LIN {X 0,Y 189.818,Z 500.496,A -85,B 0,C 180,E1 4850.971,E2 4850.971} C_VEL
LIN {X 0,Y 177.426,Z 516.785,A -85,B 0,C 180,E1 4849.524,E2 4849.524} C_VEL
LIN {X 0,Y 163.744,Z 531.874,A -85,B 0,C 180,E1 4847.674,E2 4847.674} C_VEL
LIN {X 0,Y 148.865,Z 545.693,A -85,B 0,C 180,E1 4845.27,E2 4845.27} C_VEL
LIN {X 0,Y 133.387,Z 557.829,A -85,B 0,C 180,E1 4842.163,E2 4842.163} C_VEL
LIN {X 0,Y 117.507,Z 568.332,A -85,B 0,C 180,E1 4838.035,E2 4838.035} C_VEL
LIN {X 0,Y 101.557,Z 577.191,A -85,B 0,C 180,E1 4832.376,E2 4832.376} C_VEL
LIN {X 0,Y 86.866,Z 584.067,A -85,B 0,C 180,E1 4824.801,E2 4824.801} C_VEL
LIN {X 0,Y 73.302,Z 589.412,A -85,B 0,C 180,E1 4813.7,E2 4813.7} C_VEL
LIN {X 0,Y 63.497,Z 592.778,A -85,B 0,C 180,E1 4799.212,E2 4799.212} C_VEL
LIN {X 0,Y 58.16,Z 594.477,A -85,B 0,C 180,E1 4780.894,E2 4780.894} C_VEL
LIN {X 0,Y 57.57,Z 594.636,A -85,B 0,C 180,E1 4765.012,E2 4765.012} C_VEL
LIN {X 0,Y 61.019,Z 593.564,A -85,B 0,C 180,E1 4746.836,E2 4746.836} C_VEL
LIN {X 0,Y 68.986,Z 590.981,A -85,B 0,C 180,E1 4731.442,E2 4731.442} C_VEL
LIN {X 0,Y 79.249,Z 587.223,A -85,B 0,C 180,E1 4720.526,E2 4720.526} C_VEL
LIN {X 0,Y 61.349,Z 590.587,A -85,B 0,C 180,E1 4687.494,E2 4687.494} C_VEL
LIN {X 0,Y 60.347,Z 592.025,A -85,B 0,C 180,E1 4673.342,E2 4673.342} C_VEL
LIN {X 0,Y 62.82,Z 593.696,A -85,B 0,C 180,E1 4658.528,E2 4658.528} C_VEL
LIN {X 0,Y 72.454,Z 596.219,A -85,B 0,C 180,E1 4640.504,E2 4640.504} C_VEL
LIN {X 0,Y 61.913,Z 600.596,A -85,B 0,C 180,E1 4625.554,E2 4625.554} C_VEL
LIN {X 0,Y 56.913,Z 603.196,A -85,B 0,C 180,E1 4606.332,E2 4606.332} C_VEL
LIN {X 0,Y 57.134,Z 603.987,A -85,B 0,C 180,E1 4591.009,E2 4591.009} C_VEL
LIN {X 0,Y 56.697,Z 603.74,A -85,B 0,C 180,E1 4581.896,E2 4581.896} C_VEL
LIN {X 0,Y 58.725,Z 601.943,A -85,B 0,C 180,E1 4562.639,E2 4562.639} C_VEL
LIN {X 0,Y 66.617,Z 598.284,A -85,B 0,C 180,E1 4545.144,E2 4545.144} C_VEL
LIN {X 0,Y 79.052,Z 592.754,A -85,B 0,C 180,E1 4532.077,E2 4532.077} C_VEL
LIN {X 0,Y 93.56,Z 585.667,A -85,B 0,C 180,E1 4523.221,E2 4523.221} C_VEL
LIN {X 0,Y 108.939,Z 577.083,A -85,B 0,C 180,E1 4517.079,E2 4517.079} C_VEL
LIN {X 0,Y 124.062,Z 567.359,A -85,B 0,C 180,E1 4512.807,E2 4512.807} C_VEL
LIN {X 0,Y 139.915,Z 555.487,A -85,B 0,C 180,E1 4509.459,E2 4509.459} C_VEL
LIN {X 0,Y 155.122,Z 542.173,A -85,B 0,C 180,E1 4506.984,E2 4506.984} C_VEL
LIN {X 0,Y 169.889,Z 526.958,A -85,B 0,C 180,E1 4505.064,E2 4505.064} C_VEL
LIN {X 0,Y 177.913,Z 517.465,A -85,B 0,C 180,E1 4504.176,E2 4504.176} C_VEL
LIN {X 0,Y 182.355,Z 511.668,A -85,B 0,C 180,E1 4503.395,E2 4503.395} C_VEL
LIN {X 0,Y 192.382,Z 496.615,A -85,B 0,C 180,E1 4500.658,E2 4500.658} C_VEL
LIN {X 0,Y 196.325,Z 490.237,A -85,B 0,C 180,E1 4500.079,E2 4500.079} C_VEL
LIN {X 0,Y 206.249,Z 472.484,A -85,B 0,C 180,E1 4499.444,E2 4499.444} C_VEL
LIN {X 0,Y 214.496,Z 454.315,A -85,B 0,C 180,E1 4498.981,E2 4498.981} C_VEL
LIN {X 0,Y 221.368,Z 434.904,A -85,B 0,C 180,E1 4498.629,E2 4498.629} C_VEL
LIN {X 0,Y 226.556,Z 414.734,A -85,B 0,C 180,E1 4498.331,E2 4498.331} C_VEL
LIN {X 0,Y 230.027,Z 393.555,A -85,B 0,C 180,E1 4498.043,E2 4498.043} C_VEL
LIN {X 0,Y 234.56,Z 356.946,A -85,B 0,C 180,E1 4497.556,E2 4497.556} C_VEL
LIN {X 0,Y 234.539,Z 357.104,A -85,B 0,C 180,E1 4497.279,E2 4497.279} C_VEL
LIN {X 0,Y 228.09,Z 406.713,A -85,B 0,C 180,E1 4496.629,E2 4496.629} C_VEL
LIN {X 0,Y 223.651,Z 426.828,A -85,B 0,C 180,E1 4496.277,E2 4496.277} C_VEL
LIN {X 0,Y 217.544,Z 446.236,A -85,B 0,C 180,E1 4495.807,E2 4495.807} C_VEL
LIN {X 0,Y 209.702,Z 465.163,A -85,B 0,C 180,E1 4495.188,E2 4495.188} C_VEL
LIN {X 0,Y 199.927,Z 483.847,A -85,B 0,C 180,E1 4494.376,E2 4494.376} C_VEL
LIN {X 0,Y 188.732,Z 501.277,A -85,B 0,C 180,E1 4493.36,E2 4493.36} C_VEL
LIN {X 0,Y 176.15,Z 517.521,A -85,B 0,C 180,E1 4492.076,E2 4492.076} C_VEL
LIN {X 0,Y 162.227,Z 532.577,A -85,B 0,C 180,E1 4490.432,E2 4490.432} C_VEL
LIN {X 0,Y 147.978,Z 545.6,A -85,B 0,C 180,E1 4488.432,E2 4488.432} C_VEL
LIN {X 0,Y 132.08,Z 557.864,A -85,B 0,C 180,E1 4485.678,E2 4485.678} C_VEL
LIN {X 0,Y 115.647,Z 568.483,A -85,B 0,C 180,E1 4481.985,E2 4481.985} C_VEL
LIN {X 0,Y 98.949,Z 577.451,A -85,B 0,C 180,E1 4476.849,E2 4476.849} C_VEL
LIN {X 0,Y 82.499,Z 584.718,A -85,B 0,C 180,E1 4469.363,E2 4469.363} C_VEL
LIN {X 0,Y 67.953,Z 589.994,A -85,B 0,C 180,E1 4458.617,E2 4458.617} C_VEL
LIN {X 0,Y 56.638,Z 593.427,A -85,B 0,C 180,E1 4443.171,E2 4443.171} C_VEL
LIN {X 0,Y 50.342,Z 595.123,A -85,B 0,C 180,E1 4422.612,E2 4422.612} C_VEL
LIN {X 0,Y 49.628,Z 595.281,A -85,B 0,C 180,E1 4404.211,E2 4404.211} C_VEL
LIN {X 0,Y 53.752,Z 594.211,A -85,B 0,C 180,E1 4383.478,E2 4383.478} C_VEL
LIN {X 0,Y 63.506,Z 591.436,A -85,B 0,C 180,E1 4366.144,E2 4366.144} C_VEL
LIN {X 0,Y 68.796,Z 589.752,A -85,B 0,C 180,E1 4360.217,E2 4360.217} C_VEL
LIN {X 0,Y 53.866,Z 592.475,A -85,B 0,C 180,E1 4329.619,E2 4329.619} C_VEL
LIN {X 0,Y 52.595,Z 594.013,A -85,B 0,C 180,E1 4312.355,E2 4312.355} C_VEL
LIN {X 0,Y 55.296,Z 595.519,A -85,B 0,C 180,E1 4296.561,E2 4296.561} C_VEL
LIN {X 0,Y 62.782,Z 597.31,A -85,B 0,C 180,E1 4281.136,E2 4281.136} C_VEL
LIN {X 0,Y 52.465,Z 601.062,A -85,B 0,C 180,E1 4263.559,E2 4263.559} C_VEL
LIN {X 0,Y 48.69,Z 603.014,A -85,B 0,C 180,E1 4241.858,E2 4241.858} C_VEL
LIN {X 0,Y 49.2,Z 603.359,A -85,B 0,C 180,E1 4230.007,E2 4230.007} C_VEL
LIN {X 0,Y 48.989,Z 602.601,A -85,B 0,C 180,E1 4212.181,E2 4212.181} C_VEL
LIN {X 0,Y 54.226,Z 600.219,A -85,B 0,C 180,E1 4191.186,E2 4191.186} C_VEL
LIN {X 0,Y 64.861,Z 596.198,A -85,B 0,C 180,E1 4175.224,E2 4175.224} C_VEL
LIN {X 0,Y 79.729,Z 590.089,A -85,B 0,C 180,E1 4163.739,E2 4163.739} C_VEL
LIN {X 0,Y 95.858,Z 582.41,A -85,B 0,C 180,E1 4156.353,E2 4156.353} C_VEL
LIN {X 0,Y 113.117,Z 572.703,A -85,B 0,C 180,E1 4151.163,E2 4151.163} C_VEL
LIN {X 0,Y 130.107,Z 561.376,A -85,B 0,C 180,E1 4147.564,E2 4147.564} C_VEL
LIN {X 0,Y 146.523,Z 548.432,A -85,B 0,C 180,E1 4144.968,E2 4144.968} C_VEL
LIN {X 0,Y 161.707,Z 534.309,A -85,B 0,C 180,E1 4143.105,E2 4143.105} C_VEL
LIN {X 0,Y 176.043,Z 518.521,A -85,B 0,C 180,E1 4141.675,E2 4141.675} C_VEL
LIN {X 0,Y 188.478,Z 502.268,A -85,B 0,C 180,E1 4140.646,E2 4140.646} C_VEL
LIN {X 0,Y 196.325,Z 490.237,A -85,B 0,C 180,E1 4140.079,E2 4140.079} C_VEL
LIN {X 0,Y 196.548,Z 489.749,A -85,B 0,C 180,E1 4139.711,E2 4139.711} C_VEL
LIN {X 0,Y 195.805,Z 490.724,A -85,B 0,C 180,E1 4138.944,E2 4138.944} C_VEL
LIN {X 0,Y 193.489,Z 494.15,A -85,B 0,C 180,E1 4137.813,E2 4137.813} C_VEL
LIN {X 0,Y 187.516,Z 502.681,A -85,B 0,C 180,E1 4136.334,E2 4136.334} C_VEL
LIN {X 0,Y 180.577,Z 511.792,A -85,B 0,C 180,E1 4135.192,E2 4135.192} C_VEL
LIN {X 0,Y 178.13,Z 514.759,A -85,B 0,C 180,E1 4134.93,E2 4134.93} C_VEL
LIN {X 0,Y 164.98,Z 529.345,A -85,B 0,C 180,E1 4133.655,E2 4133.655} C_VEL
LIN {X 0,Y 150.183,Z 543.194,A -85,B 0,C 180,E1 4131.962,E2 4131.962} C_VEL
LIN {X 0,Y 134.131,Z 555.801,A -85,B 0,C 180,E1 4129.711,E2 4129.711} C_VEL
LIN {X 0,Y 117.494,Z 566.709,A -85,B 0,C 180,E1 4126.716,E2 4126.716} C_VEL
LIN {X 0,Y 100.575,Z 575.897,A -85,B 0,C 180,E1 4122.612,E2 4122.612} C_VEL
LIN {X 0,Y 83.789,Z 583.36,A -85,B 0,C 180,E1 4116.746,E2 4116.746} C_VEL
LIN {X 0,Y 67.436,Z 589.214,A -85,B 0,C 180,E1 4107.674,E2 4107.674} C_VEL
LIN {X 0,Y 53.528,Z 593.182,A -85,B 0,C 180,E1 4093.71,E2 4093.71} C_VEL
LIN {X 0,Y 44.133,Z 595.395,A -85,B 0,C 180,E1 4072.643,E2 4072.643} C_VEL
LIN {X 0,Y 41.493,Z 596.021,A -85,B 0,C 180,E1 4049.991,E2 4049.991} C_VEL
LIN {X 0,Y 44.443,Z 595.358,A -85,B 0,C 180,E1 4026.102,E2 4026.102} C_VEL
LIN {X 0,Y 53.504,Z 593.24,A -85,B 0,C 180,E1 4006.247,E2 4006.247} C_VEL
LIN {X 0,Y 58.439,Z 591.929,A -85,B 0,C 180,E1 3999.803,E2 3999.803} C_VEL
LIN {X 0,Y 45.886,Z 594.249,A -85,B 0,C 180,E1 3970.042,E2 3970.042} C_VEL
LIN {X 0,Y 44.876,Z 595.756,A -85,B 0,C 180,E1 3949.735,E2 3949.735} C_VEL
LIN {X 0,Y 48.139,Z 597.165,A -85,B 0,C 180,E1 3932.813,E2 3932.813} C_VEL
LIN {X 0,Y 52.998,Z 598.262,A -85,B 0,C 180,E1 3921.805,E2 3921.805} C_VEL
LIN {X 0,Y 42.779,Z 601.446,A -85,B 0,C 180,E1 3899.404,E2 3899.404} C_VEL
LIN {X 0,Y 40.896,Z 602.619,A -85,B 0,C 180,E1 3874.215,E2 3874.215} C_VEL
LIN {X 0,Y 41.099,Z 602.684,A -85,B 0,C 180,E1 3868.615,E2 3868.615} C_VEL
LIN {X 0,Y 41.881,Z 601.681,A -85,B 0,C 180,E1 3844.559,E2 3844.559} C_VEL
LIN {X 0,Y 49.745,Z 599.007,A -85,B 0,C 180,E1 3821.965,E2 3821.965} C_VEL
LIN {X 0,Y 63.781,Z 594.326,A -85,B 0,C 180,E1 3806.034,E2 3806.034} C_VEL
LIN {X 0,Y 80.271,Z 587.905,A -85,B 0,C 180,E1 3796.458,E2 3796.458} C_VEL
LIN {X 0,Y 97.586,Z 579.806,A -85,B 0,C 180,E1 3790.411,E2 3790.411} C_VEL
LIN {X 0,Y 114.697,Z 570.227,A -85,B 0,C 180,E1 3786.423,E2 3786.423} C_VEL
LIN {X 0,Y 131.24,Z 559.231,A -85,B 0,C 180,E1 3783.648,E2 3783.648} C_VEL
LIN {X 0,Y 147.032,Z 546.849,A -85,B 0,C 180,E1 3781.641,E2 3781.641} C_VEL
LIN {X 0,Y 161.97,Z 533.054,A -85,B 0,C 180,E1 3780.152,E2 3780.152} C_VEL
LIN {X 0,Y 175.994,Z 517.747,A -85,B 0,C 180,E1 3779.013,E2 3779.013} C_VEL
LIN {X 0,Y 188.451,Z 501.615,A -85,B 0,C 180,E1 3778.175,E2 3778.175} C_VEL
LIN {X 0,Y 199.649,Z 484.197,A -85,B 0,C 180,E1 3777.535,E2 3777.535} C_VEL
LIN {X 0,Y 206.65,Z 471.197,A -85,B 0,C 180,E1 3777.185,E2 3777.185} C_VEL
LIN {X 0,Y 196.838,Z 488.697,A -85,B 0,C 180,E1 3776.471,E2 3776.471} C_VEL
LIN {X 0,Y 185.52,Z 505.346,A -85,B 0,C 180,E1 3775.574,E2 3775.574} C_VEL
LIN {X 0,Y 178.13,Z 514.759,A -85,B 0,C 180,E1 3774.93,E2 3774.93} C_VEL
LIN {X 0,Y 173.089,Z 520.671,A -85,B 0,C 180,E1 3774.797,E2 3774.797} C_VEL
LIN {X 0,Y 159.181,Z 535.058,A -85,B 0,C 180,E1 3775.604,E2 3775.604} C_VEL
LIN {X 0,Y 153.525,Z 540.284,A -85,B 0,C 180,E1 3775.428,E2 3775.428} C_VEL
LIN {X 0,Y 137.802,Z 553.027,A -85,B 0,C 180,E1 3773.715,E2 3773.715} C_VEL
LIN {X 0,Y 121.323,Z 564.182,A -85,B 0,C 180,E1 3771.454,E2 3771.454} C_VEL
LIN {X 0,Y 104.129,Z 573.818,A -85,B 0,C 180,E1 3768.336,E2 3768.336} C_VEL
LIN {X 0,Y 86.415,Z 581.898,A -85,B 0,C 180,E1 3763.795,E2 3763.795} C_VEL
LIN {X 0,Y 69.457,Z 588.057,A -85,B 0,C 180,E1 3757.102,E2 3757.102} C_VEL
LIN {X 0,Y 53.89,Z 592.467,A -85,B 0,C 180,E1 3746.594,E2 3746.594} C_VEL
LIN {X 0,Y 40.613,Z 595.359,A -85,B 0,C 180,E1 3727.975,E2 3727.975} C_VEL
LIN {X 0,Y 33.925,Z 596.544,A -85,B 0,C 180,E1 3700.174,E2 3700.174} C_VEL
LIN {X 0,Y 34.674,Z 596.476,A -85,B 0,C 180,E1 3673.229,E2 3673.229} C_VEL
LIN {X 0,Y 42.864,Z 594.979,A -85,B 0,C 180,E1 3647.421,E2 3647.421} C_VEL
LIN {X 0,Y 48.136,Z 593.861,A -85,B 0,C 180,E1 3639.391,E2 3639.391} C_VEL
LIN {X 0,Y 37.652,Z 595.852,A -85,B 0,C 180,E1 3609.171,E2 3609.171} C_VEL
LIN {X 0,Y 37.109,Z 597.133,A -85,B 0,C 180,E1 3587.556,E2 3587.556} C_VEL
LIN {X 0,Y 41.66,Z 598.585,A -85,B 0,C 180,E1 3566.498,E2 3566.498} C_VEL
LIN {X 0,Y 43.125,Z 598.924,A -85,B 0,C 180,E1 3562.572,E2 3562.572} C_VEL
LIN {X 0,Y 33.879,Z 601.304,A -85,B 0,C 180,E1 3536.288,E2 3536.288} C_VEL
LIN {X 0,Y 33.171,Z 602.062,A -85,B 0,C 180,E1 3510.011,E2 3510.011} C_VEL
LIN {X 0,Y 34.357,Z 601.106,A -85,B 0,C 180,E1 3480.36,E2 3480.36} C_VEL
LIN {X 0,Y 44.72,Z 598.323,A -85,B 0,C 180,E1 3453.98,E2 3453.98} C_VEL
LIN {X 0,Y 60.328,Z 593.745,A -85,B 0,C 180,E1 3439.164,E2 3439.164} C_VEL
LIN {X 0,Y 78.328,Z 587.229,A -85,B 0,C 180,E1 3430.637,E2 3430.637} C_VEL
LIN {X 0,Y 96.434,Z 579.125,A -85,B 0,C 180,E1 3425.567,E2 3425.567} C_VEL
LIN {X 0,Y 114.068,Z 569.54,A -85,B 0,C 180,E1 3422.296,E2 3422.296} C_VEL
LIN {X 0,Y 130.974,Z 558.533,A -85,B 0,C 180,E1 3420.047,E2 3420.047} C_VEL
LIN {X 0,Y 147.027,Z 546.135,A -85,B 0,C 180,E1 3418.437,E2 3418.437} C_VEL
LIN {X 0,Y 162.156,Z 532.316,A -85,B 0,C 180,E1 3417.253,E2 3417.253} C_VEL
LIN {X 0,Y 168.807,Z 525.467,A -85,B 0,C 180,E1 3416.811,E2 3416.811} C_VEL
LIN {X 0,Y 154.443,Z 539.446,A -85,B 0,C 180,E1 3415.518,E2 3415.518} C_VEL
LIN {X 0,Y 153.525,Z 540.284,A -85,B 0,C 180,E1 3415.428,E2 3415.428} C_VEL
LIN {X 0,Y 146.896,Z 546.017,A -85,B 0,C 180,E1 3415.143,E2 3415.143} C_VEL
LIN {X 0,Y 129.682,Z 558.869,A -85,B 0,C 180,E1 3415.731,E2 3415.731} C_VEL
LIN {X 0,Y 121.836,Z 563.938,A -85,B 0,C 180,E1 3415.403,E2 3415.403} C_VEL
LIN {X 0,Y 121.319,Z 564.266,A -85,B 0,C 180,E1 3415.343,E2 3415.343} C_VEL
LIN {X 0,Y 103.779,Z 573.977,A -85,B 0,C 180,E1 3412.88,E2 3412.88} C_VEL
LIN {X 0,Y 86.432,Z 581.768,A -85,B 0,C 180,E1 3409.488,E2 3409.488} C_VEL
LIN {X 0,Y 68.581,Z 588.126,A -85,B 0,C 180,E1 3404.181,E2 3404.181} C_VEL
LIN {X 0,Y 50.77,Z 592.92,A -85,B 0,C 180,E1 3394.93,E2 3394.93} C_VEL
LIN {X 0,Y 35.312,Z 595.902,A -85,B 0,C 180,E1 3377.392,E2 3377.392} C_VEL
LIN {X 0,Y 26.318,Z 597.17,A -85,B 0,C 180,E1 3345.408,E2 3345.408} C_VEL
LIN {X 0,Y 26.553,Z 597.159,A -85,B 0,C 180,E1 3312.453,E2 3312.453} C_VEL
LIN {X 0,Y 35.971,Z 595.837,A -85,B 0,C 180,E1 3281.352,E2 3281.352} C_VEL
LIN {X 0,Y 37.448,Z 595.611,A -85,B 0,C 180,E1 3278.405,E2 3278.405} C_VEL
LIN {X 0,Y 29.431,Z 597.189,A -85,B 0,C 180,E1 3247.814,E2 3247.814} C_VEL
LIN {X 0,Y 32.744,Z 599.172,A -85,B 0,C 180,E1 3206.662,E2 3206.662} C_VEL
LIN {X 0,Y 33.38,Z 599.344,A -85,B 0,C 180,E1 3203.991,E2 3203.991} C_VEL
LIN {X 0,Y 24.863,Z 601.158,A -85,B 0,C 180,E1 3166.365,E2 3166.365} C_VEL
LIN {X 0,Y 25.005,Z 601.388,A -85,B 0,C 180,E1 3148.343,E2 3148.343} C_VEL
LIN {X 0,Y 27.991,Z 600.357,A -85,B 0,C 180,E1 3110.004,E2 3110.004} C_VEL
LIN {X 0,Y 40.611,Z 597.672,A -85,B 0,C 180,E1 3084.387,E2 3084.387} C_VEL
LIN {X 0,Y 58.14,Z 593.072,A -85,B 0,C 180,E1 3071.437,E2 3071.437} C_VEL
LIN {X 0,Y 77.23,Z 586.554,A -85,B 0,C 180,E1 3064.588,E2 3064.588} C_VEL
LIN {X 0,Y 96.283,Z 578.301,A -85,B 0,C 180,E1 3060.594,E2 3060.594} C_VEL
LIN {X 0,Y 115.234,Z 568.143,A -85,B 0,C 180,E1 3058.01,E2 3058.01} C_VEL
LIN {X 0,Y 131.175,Z 557.872,A -85,B 0,C 180,E1 3056.448,E2 3056.448} C_VEL
LIN {X 0,Y 121.319,Z 564.266,A -85,B 0,C 180,E1 3055.343,E2 3055.343} C_VEL
LIN {X 0,Y 113.22,Z 569.107,A -85,B 0,C 180,E1 3054.803,E2 3054.803} C_VEL
LIN {X 0,Y 95.57,Z 578.083,A -85,B 0,C 180,E1 3055.117,E2 3055.117} C_VEL
LIN {X 0,Y 85.594,Z 582.33,A -85,B 0,C 180,E1 3054.743,E2 3054.743} C_VEL
LIN {X 0,Y 82.51,Z 583.556,A -85,B 0,C 180,E1 3054.296,E2 3054.296} C_VEL
LIN {X 0,Y 62.999,Z 589.943,A -85,B 0,C 180,E1 3049.703,E2 3049.703} C_VEL
LIN {X 0,Y 44.265,Z 594.356,A -85,B 0,C 180,E1 3041.542,E2 3041.542} C_VEL
LIN {X 0,Y 27.372,Z 596.973,A -85,B 0,C 180,E1 3023.454,E2 3023.454} C_VEL
LIN {X 0,Y 17.951,Z 597.874,A -85,B 0,C 180,E1 2982.853,E2 2982.853} C_VEL
LIN {X 0,Y 20.894,Z 597.669,A -85,B 0,C 180,E1 2934.931,E2 2934.931} C_VEL
LIN {X 0,Y 26.885,Z 597.079,A -85,B 0,C 180,E1 2916.99,E2 2916.99} C_VEL
LIN {X 0,Y 20.946,Z 598.607,A -85,B 0,C 180,E1 2874.527,E2 2874.527} C_VEL
LIN {X 0,Y 23.786,Z 599.562,A -85,B 0,C 180,E1 2846.882,E2 2846.882} C_VEL
LIN {X 0,Y 16.997,Z 600.754,A -85,B 0,C 180,E1 2790.647,E2 2790.647} C_VEL
LIN {X 0,Y 21.688,Z 599.78,A -85,B 0,C 180,E1 2738.425,E2 2738.425} C_VEL
LIN {X 0,Y 37.956,Z 597.003,A -85,B 0,C 180,E1 2712.964,E2 2712.964} C_VEL
LIN {X 0,Y 57.078,Z 592.4,A -85,B 0,C 180,E1 2703.266,E2 2703.266} C_VEL
LIN {X 0,Y 77.011,Z 585.878,A -85,B 0,C 180,E1 2698.434,E2 2698.434} C_VEL
LIN {X 0,Y 93.205,Z 579.207,A -85,B 0,C 180,E1 2696.02,E2 2696.02} C_VEL
LIN {X 0,Y 82.51,Z 583.556,A -85,B 0,C 180,E1 2694.296,E2 2694.296} C_VEL
LIN {X 0,Y 74.148,Z 586.638,A -85,B 0,C 180,E1 2693.395,E2 2693.395} C_VEL
LIN {X 0,Y 54.887,Z 592.3,A -85,B 0,C 180,E1 2693.717,E2 2693.717} C_VEL
LIN {X 0,Y 44.863,Z 594.512,A -85,B 0,C 180,E1 2692.683,E2 2692.683} C_VEL
LIN {X 0,Y 43.021,Z 594.884,A -85,B 0,C 180,E1 2692.105,E2 2692.105} C_VEL
LIN {X 0,Y 24.407,Z 597.515,A -85,B 0,C 180,E1 2680.382,E2 2680.382} C_VEL
LIN {X 0,Y 10.724,Z 598.5,A -85,B 0,C 180,E1 2637.748,E2 2637.748} C_VEL
LIN {X 0,Y 13.62,Z 598.413,A -85,B 0,C 180,E1 2562.727,E2 2562.727} C_VEL
LIN {X 0,Y 16.181,Z 598.227,A -85,B 0,C 180,E1 2553.797,E2 2553.797} C_VEL
LIN {X 0,Y 13.976,Z 599.544,A -85,B 0,C 180,E1 2492.671,E2 2492.671} C_VEL
LIN {X 0,Y 8.932,Z 600.101,A -85,B 0,C 180,E1 2430.041,E2 2430.041} C_VEL
LIN {X 0,Y 18.829,Z 599.014,A -85,B 0,C 180,E1 2355.391,E2 2355.391} C_VEL
LIN {X 0,Y 38,Z 596.15,A -85,B 0,C 180,E1 2339.997,E2 2339.997} C_VEL
LIN {X 0,Y 54.426,Z 592.484,A -85,B 0,C 180,E1 2335.47,E2 2335.47} C_VEL
LIN {X 0,Y 43.021,Z 594.884,A -85,B 0,C 180,E1 2332.105,E2 2332.105} C_VEL
LIN {X 0,Y 33.473,Z 596.609,A -85,B 0,C 180,E1 2329.358,E2 2329.358} C_VEL
LIN {X 0,Y 18.738,Z 598.45,A -85,B 0,C 180,E1 2326.925,E2 2326.925} C_VEL
LIN {X 0,Y 3.35,Z 599.24,A -85,B 0,C 180,E1 2305.721,E2 2305.721} C_VEL
LIN {X 0,Y 2.717,Z 599.21,A -85,B 0,C 180,E1 2195.731,E2 2195.731} C_VEL
LIN {X 0,Y 5.275,Z 599.171,A -85,B 0,C 180,E1 2173.735,E2 2173.735} C_VEL
LIN {X 0,Y 5.008,Z 599.263,A -85,B 0,C 180,E1 2161.752,E2 2161.752} C_VEL
LIN {X 0,Y 0.825,Z 599.445,A -85,B 0,C 180,E1 2070.445,E2 2070.445} C_VEL
LIN {X 0,Y 9.86,Z 599.058,A -85,B 0,C 180,E1 1972.725,E2 1972.725} C_VEL
LIN {X 0,Y 2.717,Z 599.21,A -85,B 0,C 180,E1 1835.731,E2 1835.731} C_VEL
LIN {X 0,Y 4.517,Z 601.21,A -85,B 0,C 180,E1 1819.913,E2 1819.913} C_VEL
LIN {X 0,Y 4.517,Z 647,A -85,B 0,C 180,E1 1819.913,E2 1819.913} C_VEL
LIN {X 0,Y 4.517,Z 647,A -85,B 0,C 180,E1 1819.913,E2 1819.913}

QRS_NEXT_CUT()

QRS_NEXT()
QRS_HOME()

END
